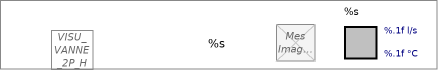
VISUALIZATION VISU_LIGNE_EAU_FLOWTEMP  // 438x70
VAR_IN_OUT
	m_Input_LIGNE_EAU : BLOCK_LIGNE_REF_FLOWTEMP;
END_VAR
    Polyline (451,20)
    Polyline (80,20)
    Polyline (129,20)
    Polygon (140,20)
    Polygon (317,20)
    Rectangle (154,28 125x31), "%s", text variable: m_Input_LIGNE_EAU.mnemo
    Frame (51,30 42x40)
        shows VISU_VANNE_2P_H(m_Input_VANNE := m_Input_LIGNE_EAU.VEx)
        p1022016623: m_Input_LIGNE_EAU.VEx
    Image (276,24 39x37), invisible if: NOT m_Input_LIGNE_EAU.STATE_NOK, image: MesImages.warning
    Rectangle (381,23 45x15), "%.1f l/s", text variable: m_Input_LIGNE_EAU.DEx.STATE_Flow, invisible if: m_Input_LIGNE_EAU.CONF_Max_Flow = 0 AND m_Input_LIGNE_EAU.CONF_Min_Flow = 0
    Rectangle (341,0 36x23), "%s", text variable: m_Input_LIGNE_EAU.mnemo_DEX
    Rectangle (344,26 33x33), colour toggle: m_Input_LIGNE_EAU.STATE_DexT AND m_Input_LIGNE_EAU.VEx.STATE_On
    Polyline (16,8)
    Polyline (24,15)
    Rectangle (381,46 45x15), "%.1f °C", text variable: m_Input_LIGNE_EAU.DEx.STATE_Temp
END_VISUALIZATION

(* stored: Version 1.1.0.1, ProductVersion 3.1.4024.12
   Visu VISU_LIGNE_EAU_FLOWTEMP: Id {e0950b9e-2e9f-45bc-b3e8-e7f87055b3d0} *)
